// TIA Portal V17 export
// export: Created 2021-12-03T08:12:52.4232354Z, ExportSetting WithDefaults, DisplayName Totally Integrated Automation Portal, DisplayVersion V17, DisplayName TIA Portal Openness, DisplayVersion V17, DisplayName TIA Portal Version Control Interface, DisplayVersion V17, DisplayName STEP 7 Professional, DisplayVersion V17, DisplayName STEP 7 Safety, DisplayVersion V17, DisplayName WinCC Advanced, DisplayVersion V17
DATA_BLOCK "GDB_HMI_Data"   // DB1001
VERSION : 0.1
// stored: AutoNumber false, IsOnlyStoredInLoadMemory false, IsWriteProtectedInAS false
   VAR
      Receive : Struct
         CmndOn : Struct   // Команды на включение/запуска
            bit00_Pwr : Bool;   // Подача питания на все элементы
            bit01_FrqConvPwr : Bool;   // Подача питания на частотный преобразователь
            bit02_SrvcMd : Bool;   // Сервисный режим
            bit03_PwrAcc : Bool;   // Питание ускорителя
            bit04 : Bool;
            bit05 : Bool;
            bit06 : Bool;
            bit07 : Bool;
            bit08 : Bool;
            bit09 : Bool;
            bit10 : Bool;
            bit11 : Bool;
            bit12 : Bool;
            bit13 : Bool;
            bit14 : Bool;
            bit15 : Bool;
         END_STRUCT;
         CmndOff : Struct   // Команды на выключение/останов
            bit00_Pwr : Bool;   // Общее отключение питания
            bit01_FrqConvPwr : Bool;   // Отключение питания на частотном преобразователе
            bit02_SrvcMd : Bool;   // Сервисный режим
            bit03_PwrAcc : Bool;   // Питание ускорителя
            bit04 : Bool;
            bit05 : Bool;
            bit06 : Bool;
            bit07 : Bool;
            bit08 : Bool;
            bit09 : Bool;
            bit10 : Bool;
            bit11 : Bool;
            bit12 : Bool;
            bit13 : Bool;
            bit14 : Bool;
            bit15 : Bool;
         END_STRUCT;
         Cmnd_AckRst : Struct   // Команды сброс/подтверждение
            bit00_Faults : Bool;   // Сброс/ квитирование ошибок
            bit01_AccFaults : Bool;   // Сброс ошибок ускорителя
            bit02_AccFullWrmUp : Bool;   // Прогрев после паузы
            bit03_AccPwrRst : Bool;   // Сброс питания ускорителя
            bit04_DetLinePwrRst : Bool;   // Сброс питания линейки
            bit05_ParDefltRst : Bool;   // Сброс параметров к заводским настройкам для гантри
            bit06_WarmUpFull : Bool;
            bit07_StrtScan : Bool;
            bit08_StpScan : Bool;
            bit09 : Bool;
            bit10 : Bool;
            bit11 : Bool;
            bit12 : Bool;
            bit13 : Bool;
            bit14 : Bool;
            bit15 : Bool;
            bit16 : Bool;
            bit17 : Bool;
            bit18 : Bool;
            bit19 : Bool;
            bit20 : Bool;
            bit21 : Bool;
            bit22 : Bool;
            bit23 : Bool;
            bit24 : Bool;
            bit25 : Bool;
            bit26 : Bool;
            bit27 : Bool;
            bit28 : Bool;
            bit29 : Bool;
            bit30 : Bool;
            bit31 : Bool;
         END_STRUCT;
         CmndSwitch : Struct   // Команды переключений
            bit00_FastOnAcc : Bool;   // Быстрое включение
            bit01_FastOffAcc : Bool;   // Быстрое отключение
            bit02_ : Bool;
            bit03_ : Bool;
            bit04_ : Bool;
            bit05_ : Bool;
            bit06_ : Bool;
            bit07_ : Bool;
            bit08_ : Bool;
            bit09_ : Bool;
            bit10_ : Bool;
            bit11_ : Bool;
            bit12_ : Bool;
            bit13_ : Bool;
            bit14_ : Bool;
            bit15_ : Bool;
         END_STRUCT;
         Simulation : Struct   // Симуляция
            PSConv_SimEn : Bool;   // Симуляция фотосенсеров
            Acc_SimEn : Bool;   // Симуляция сигналов ускорителя
            Console_SimEn : Bool;   // Симуляция панели управления
            AccChilSwitch_SimEn : Bool;   // Симуляция переключения чиллела и модулятора
            PrDor_SimEn : Bool;   // Симуляция защитной двери
            EmSt_SimEn : Bool;   // Симуляция авариных кнопок
            FBPower_SimEn : Bool;   // Симуляция контакторов обратная связь
            Power_SimEn : Bool;   // Симуляция питания
            FrConv_SimEn : Bool;   // Симуляция преобразователя частоты
            EmStp : Struct
               "/AccCon_Ch1" : Bool;   // Консоль ускорителя канал 1
               "/P1_Ch1" : Bool;   // Пульт Р1 канал 1
               "/P2_Ch1" : Bool;   // Пульт Р2 канал 1
               "/Dosimeter_Ch1" : Bool;   // Дозиметр канал 1
               "/P3_Ch1" : Bool;   // Пульт P3 канал 1
               Com : Bool;   // Общая
            END_STRUCT;
            PrDoor : Struct
               PrDoor1Cls_Ch1 : Bool;   // Замок блокирующий дверь 1 канал 1
               PrDoor2Cls_Ch1 : Bool;   // Замок блокирующий дверь 2 канал 1
               PrDoor1Req : Bool;   // Запрос на открытие двери 1
               PrDoor2Req : Bool;   // Запрос на открытие двери 2
            END_STRUCT;
            SupplyChains : Struct
               Com : Bool;   // Simulation Breaker All
               BrLigSrvFlt : Bool;   // Simulation Breaker Light and Service Outlet Fault
               BrModFlt : Bool;   // Simulation Breaker Modulator Fault
               BrChilFlt : Bool;   // Simulation Breaker Chiller Fault
               BrPow1Flt : Bool;   // Simulation Breaker Powersupply 1 24VDC Fault
               BrPow2Flt : Bool;   // Simulation Breaker Powersupply 2 24VDC Fault
               BrFrqConvFlt : Bool;   // Simulation Breaker Frequnce Converter Conveyor Fault
               BrAccConFlt : Bool;   // Simulation Breaker Accelerator Console Fault
               BrXRayUnitFlt : Bool;   // Simulation Breaker X-Ray Unit Fault
               BrPowPlcFlt : Bool;   // Simulation Breaker Powersupply PS307 (PLC) Fault
               SitopPow1Flt : Bool;   // Simulation Sitop Diagnose Modul Powersupply 1 Failure
               SitopPow2Flt : Bool;   // Simulation Sitop Diagnose Modul Powersupply 2 Failure
               BrMod1PFlt : Bool;   // Simulation Breaker Modulator 230 VAC Fault
            END_STRUCT;
            ScanSeq : Struct
               DetLineRdy : Bool;   // Готовность детекторной линейки
            END_STRUCT;
            Console : Struct
               P2 : Bool;
               P2ConvLocal : Bool;   // Simulation Panel 2: Keyswitch Conveyor Local
               "/P2ConvLocal" : Bool;   // Simulation Panel 2: Keyswitch Conveyor Local (False=Local)
               P2ConvFwd : Bool;   // Simulation Panel 2: Conveyor move forward
               P2ConvBwd : Bool;   // Simulation Panel 2: Conveyor move backward
               P3AckInSArea_Ch1 : Bool;   // Сброс внутри периметра безопасности
               P1AckEmStpOutSArea : Bool;   // Сброс снаружи периметра безопасности
               P2AgreeBut_Ch1 : Bool;   // Кнопка разрешения канал 1
               P1KeyGenRel_Ch1 : Bool;   // Главный ключ разрешения канал 1
               P1KeyAccRel_Ch1 : Bool;   // Ключ разрешения включения ускорителя канал 1
            END_STRUCT;
            PhotoSensor : Struct
               PSConvStpBwd : Bool;   // Simulation Photo Sensor Conveyor Stop Position Back
               PSConvSlowBwd : Bool;   // Simulation Photo Sensor Conveyor Fast Slow Back
               PSConvSlowFwd : Bool;   // Simulation Photo Sensor Conveyor Fast Slow Front
               PSConvStpFwd : Bool;   // Simulation Photo Sensor Conveyor Stop Position Front
               PSConvXRayBwd : Bool;   // Simulation Photo Sensor Conveyor Sensor X-Ray Back
               PSConvXRayFwd : Bool;   // Simulation Photo Sensor Conveyor Sensor X-Ray Front
            END_STRUCT;
            AccChilSwitch : Struct
               ChilVlv_Acc1_Pos : Bool;   // Simulation Chiller Valve Position 1
               ChilVlv_Acc2_Pos : Bool;   // Simulation Chiller Valve Position 2
               ModSwch_Acc1_Pos : Bool;   // Simulation Modulator Switch Position 1
               ModSwch_Acc2_Pos : Bool;   // Simulation Modulator Switch Position 2
            END_STRUCT;
            Acc : Struct
               AccStRemMode : Bool;   // Simulation Accelerator Status: Remote Mode selected
               AccStPowerOn : Bool;   // Simulation Accelerator Status: Power on
               AccStWarmUp : Bool;   // Simulation Accelerator Status: Warming up
               AccStClear : Bool;   // Simulation Accelerator Status: Clear
               AccStReady : Bool;   // Simulation Accelerator Status: Ready
               AccStXRayOn : Bool;   // Simulation Accelerator Status: X-Ray on
               AccStFault : Bool;   // Simulation Accelerator Status: Fault
               AccStNoEmStp : Bool;   // Simulation Accelerator Status: Emergency Stop not active
               AccStStandby : Bool;   // Simulation Accelerator Status: Standby
               AccStMicroWave : Bool;   // Simulation Accelerator Status: Microwave (TIS, MIS)
               AccStHighDoze : Bool;   // Simulation Accelerator Status: High Doze (MIS)
               AccStRemouteKey : Bool;   // Simulation Accelerator Status: Acc Panel Key
               AccStEmStpPanel : Bool;   // Simulation Accelerator Status: Emergency Stop Panel (True=No EmStp)
            END_STRUCT;
         END_STRUCT;
      END_STRUCT;
   END_VAR
BEGIN
END_DATA_BLOCK
